FUNCTION_BLOCK TcoEvaluateMeasurementTask EXTENDS TcoCore.TcoRemoteTask
VAR

	_config:TcoEvaluateMeasurementConfig;

	_data : ARRAY [0..1000] OF TcoEvaluateMeasurementDataItem;	
	
	_results:TcoEvaluateMeasurementResults;
	_entityId: STRING;
	{attribute 'hide'}
	_cleanResultData: TcoEvaluateMeasurementResults;
	{attribute 'hide'}
	_cleanData:ARRAY [0..1000] OF TcoEvaluateMeasurementDataItem;	
END_VAR

SUPER^();

PROPERTY Config : TcoEvaluateMeasurementConfig
GET
Config:=_config;
END_GET
END_PROPERTY

PROPERTY DataSource : ARRAY [0..1000] OF TcoEvaluateMeasurementDataItem
GET
DataSource:=_data;
END_GET
SET
_data:=DataSource;
END_SET
END_PROPERTY

(*~
	<docu>
		<summary>
			Restores this instance to the Ready state. Can be called explicitly or from within one of the restore mechanisms.
			<para>
				See also <see cref="PlcDocu.TcoCore.TcoTask.AutoRestorable()"/>
			</para>
		</summary>			
	</docu>	
~*)
METHOD Restore : ITcoRestorable
SUPER^.Restore();
_data:=_cleanData;
_results:=_cleanResultData;
END_METHOD

PROPERTY Results : TcoEvaluateMeasurementResults
GET
Results:=_results;
END_GET
END_PROPERTY

METHOD Run : REFERENCE TO TcoEvaluateMeasurementTask
VAR_INPUT
	inEntityId:STRING;
	inConfig:TcoEvaluateMeasurementConfig;
	inData:ARRAY [0..1000] OF TcoEvaluateMeasurementDataItem;
END_VAR
VAR
	_cleanResultData: TcoEvaluateMeasurementResults;
END_VAR
_config:=inConfig;
_entityId:=inEntityId;
_data:=inData;
Run REF= THIS^;
END_METHOD

END_FUNCTION_BLOCK

(* stored: Version 1.1.0.1, ProductVersion 3.1.4024.10
   POU TcoEvaluateMeasurementTask: Id {a7d31628-dd32-0371-02be-834276f1ff70}, SpecialFunc None
   Property Config: Id {f21403a9-4372-0fa8-354b-e0048f19bc3b}
   Get Get: Id {66f5a70b-dd23-03c9-1a01-0dd236d1aa5e}
   Property DataSource: Id {d9eaf964-d5df-0b2e-3c23-6b579777e692}
   Get Get: Id {46421f0e-7ec9-0319-3c86-eda9d8d6d9c2}
   Set Set: Id {85989d64-f1f5-02ef-2043-50e6d81b9757}
   Method Restore: Id {d85ed7e5-3791-0916-3f74-32e2aeca06b8}
   Property Results: Id {27932ba0-4326-020e-1a79-4b1162db5f99}
   Get Get: Id {13c1d3cc-0611-0713-0c6f-6bc02c3eec61}
   Method Run: Id {be7634c6-026d-0c91-1e95-5f0249c2c852} *)
